FUNCTION_BLOCK FB_ValveMock IMPLEMENTS I_Valve
VAR_INPUT
END_VAR
VAR_OUTPUT
END_VAR
VAR
    bOpenCalled : BOOL;
    bCloseCalled : BOOL;
END_VAR

{warning 'add method implementation '}
METHOD M_ActClose : BOOL (*Closes the Valve*)
    bCloseCalled := TRUE;
    M_ActClose := TRUE;
END_METHOD

{warning 'add method implementation '}
METHOD M_ActOpen : BOOL (*Opens the Valve*)
    bOpenCalled := TRUE;
    M_ActOpen := TRUE;
END_METHOD

{warning 'add method implementation '}
METHOD M_DeviceEnable : BOOL
END_METHOD

{warning 'add method implementation '}
METHOD M_DeviceHeartbeat : BOOL
END_METHOD

{warning 'add method implementation '}
METHOD M_DeviceReset : BOOL
 	bOpenCalled := FALSE;
    bCloseCalled := FALSE;
END_METHOD

{warning 'add method implementation '}
METHOD M_DeviceStatus : E_StatusFieldDevice
END_METHOD

PROPERTY pActCloseComp : BOOL
GET
END_GET
SET
END_SET
END_PROPERTY

PROPERTY pActClosedPosSensor : BOOL
SET
END_SET
END_PROPERTY

PROPERTY pActCloseOut : BOOL
GET
END_GET
SET
END_SET
END_PROPERTY

PROPERTY pActOpenComp : BOOL
GET
END_GET
SET
END_SET
END_PROPERTY

PROPERTY pActOpenedPosSensor : BOOL
SET
END_SET
END_PROPERTY

PROPERTY pActOpenOut : BOOL
GET
END_GET
SET
END_SET
END_PROPERTY

PROPERTY pDeviceCommOK : BOOL
GET
END_GET
SET
END_SET
END_PROPERTY

PROPERTY pDeviceEnableCmd : BOOL
GET
END_GET
SET
END_SET
END_PROPERTY

PROPERTY pDeviceEnabled : BOOL
GET
END_GET
SET
END_SET
END_PROPERTY

PROPERTY pDeviceFaulted : BOOL
GET
END_GET
SET
END_SET
END_PROPERTY

PROPERTY pDeviceReset : BOOL
SET
END_SET
END_PROPERTY

PROPERTY pDeviceStatusFeedback : DWORD
GET
END_GET
SET
END_SET
END_PROPERTY

END_FUNCTION_BLOCK

(* stored: Version 1.1.0.1, ProductVersion 3.1.4024.15
   POU FB_ValveMock: Id {1fa8c906-d145-4426-95fe-854ca40b457b}, SpecialFunc None
   Method M_ActClose: Id {ee444a59-c132-4658-9e9f-dee98f6c4d88}
   Method M_ActOpen: Id {8fca511c-538a-4f2a-853c-e17c0fac895e}
   Method M_DeviceEnable: Id {c8b37b27-8724-43dd-95e9-ee638ac792fa}
   Method M_DeviceHeartbeat: Id {46ad4331-73bb-4446-a51c-351cf6c8fd77}
   Method M_DeviceReset: Id {e78b3636-328a-48de-ad45-d89a16246b40}
   Method M_DeviceStatus: Id {6bcd884b-c036-4c10-bce9-88a2fe7e8796}
   Property pActCloseComp: Id {90ef72ff-dd67-488e-a3a5-cc821ba3981b}
   Get Get: Id {d9c5fdbb-e219-4961-8878-39fec21476e5}
   Set Set: Id {85513885-5c54-4be0-83b8-1ef3b06c8332}
   Property pActClosedPosSensor: Id {5cdea73f-3580-4098-bf40-d2f062f20488}
   Set Set: Id {3915627c-61f2-48eb-bd6f-aba7941ec046}
   Property pActCloseOut: Id {f5dcd3d0-b458-4b70-bdbe-d8c163b15df0}
   Get Get: Id {6566deca-91da-4631-b302-26230a379ca4}
   Set Set: Id {ffbb7095-109a-4713-b203-88f2789a8359}
   Property pActOpenComp: Id {f2d280a2-9d6e-4966-923b-f5ae482f909c}
   Get Get: Id {2ddc636b-a48a-4b5f-ae17-78de2b172de1}
   Set Set: Id {832d7ac9-6849-4f8b-8cce-b4e37f3e43fe}
   Property pActOpenedPosSensor: Id {593f2643-d7b0-45ee-85cc-5159907c42bd}
   Set Set: Id {1c441899-605d-433c-8248-0397322629a8}
   Property pActOpenOut: Id {a39bcd44-cc36-4b78-b662-38fa44e07190}
   Get Get: Id {20e0e9f4-e0af-4cda-a123-69fd9f591965}
   Set Set: Id {d3802aae-a73f-4dcd-b590-3cd7d3c6ec32}
   Property pDeviceCommOK: Id {00c70a1d-45b3-4fef-9d5c-df95d60cc0ac}
   Get Get: Id {46f48900-5392-43e8-8c95-b81220c2d51f}
   Set Set: Id {1f2659ad-8bf9-4a5e-ae8e-c62b1fd44668}
   Property pDeviceEnableCmd: Id {ede025cf-8032-4438-8174-f52dfa65619b}
   Get Get: Id {dd83f4a1-db6a-42dd-aee5-489e6f9c5282}
   Set Set: Id {5006279a-58c2-4dc0-bc70-d6af746852ec}
   Property pDeviceEnabled: Id {140dc4fa-d179-4239-90f3-5b07e45fcec6}
   Get Get: Id {3b7fcfa0-c28b-4153-8cb5-d70ed187f51f}
   Set Set: Id {4f4e7912-1d3c-4c72-b264-2be3f1943624}
   Property pDeviceFaulted: Id {e09d199e-39d6-439a-8c6c-9c3f30ad30e4}
   Get Get: Id {b24053dd-ba7e-474b-b468-153ede085680}
   Set Set: Id {6904c3fd-5e16-4927-ac39-e36b603c5abe}
   Property pDeviceReset: Id {da4469e4-a0d0-4125-b50f-ff059ecfd822}
   Set Set: Id {3fcb01b3-a6cf-4a9a-a7b1-dc808415828f}
   Property pDeviceStatusFeedback: Id {7044f426-1541-4bdd-9801-28d99ddcd296}
   Get Get: Id {83165745-0d5d-4151-945f-9f03a3c182b3}
   Set Set: Id {8adf0546-6aac-43d4-933f-c6397bf1d680} *)
